// TwinCAT 3 PLC project PlcGenerated
// ProgramVersion: 3.1.4023.0
// libraries:
//   Tc2_Standard, * (Beckhoff Automation GmbH)
//   Tc2_System, * (Beckhoff Automation GmbH)
//   Tc3_Module, * (Beckhoff Automation GmbH)
//   Tc2_EtherCAT,newest,Beckhoff Automation GmbH
// project tree:
//   DUTs/ EthercatDevice.TcDUT
//   / PlcTask.TcTTO
//   POUs/ MAIN.TcPOU
// real-time tasks:
//   TASK PlcTask: cycle T#10ms, priority 20, ADS port 350
// I/O:
//   DEVICE Device_1, AmsNetId 192.168.18.153.2.1
//     Box 1 (LAN9255_EtherCAT_Slave) [LAN9255_EtherCAT_Slave]
// variable links:
//   PlcGenerated/PlcGenerated Instance <-> Device_1/Box 1 (LAN9255_EtherCAT_Slave)
//     PlcTask Inputs/MAIN.DeviceStatus <-> Inputs process data mapping/DeviceStatus
//     PlcTask Inputs/MAIN.MotorDiagnostic <-> Inputs process data mapping/MotorDiagnostic
//     PlcTask Inputs/MAIN.mDiag3 <-> Inputs process data mapping/Diag3
//     PlcTask Inputs/MAIN.mPosition <-> Inputs process data mapping/Position
//     PlcTask Inputs/MAIN.mTemperature <-> Inputs process data mapping/Temperature
//     PlcTask Outputs/MAIN.device[1].mDirection <-> Outputs process data mapping/Direction
//     PlcTask Outputs/MAIN.device[1].mDisplacement <-> Outputs process data mapping/Displacement
//     PlcTask Outputs/MAIN.device[1].mMode <-> Outputs process data mapping/Mode
//     PlcTask Outputs/MAIN.device[1].mRPM <-> Outputs process data mapping/RPM
//     PlcTask Outputs/MAIN.device[1].mRampDelay <-> Outputs process data mapping/RampDelay
//     PlcTask Outputs/MAIN.device[1].mTime <-> Outputs process data mapping/Time

CONFIGURATION PlcGenerated
    RESOURCE PLC ON TwinCAT3
        TASK PlcTask(INTERVAL := T#10ms, PRIORITY := 20);
        PROGRAM MAIN WITH PlcTask : MAIN;
    END_RESOURCE
END_CONFIGURATION

// ---- DUTs/EthercatDevice.TcDUT
TYPE EthercatDevice :
STRUCT
    mDirection AT %Q*: BOOL;
    mRPM AT %Q*: REAL;
    mDisplacement AT %Q*: REAL;
    mTime AT %Q*: REAL;
    mRampDelay AT %Q*: REAL;
    mMode AT %Q*: DWORD;
END_STRUCT
END_TYPE

// ---- POUs/MAIN.TcPOU
PROGRAM MAIN 
VAR CONSTANT 
deviceCount : WORD := 1; 
END_VAR 
VAR 
{attribute 'TcLinkTo' := '[1].mDirection :=  TIID^Device_1^Box 1 (LAN9255_EtherCAT_Slave)^Outputs process data mapping^Direction; 
[1].mDisplacement := TIID^Device_1^Box 1 (LAN9255_EtherCAT_Slave)^Outputs process data mapping^Displacement; 
[1].mRPM := TIID^Device_1^Box 1 (LAN9255_EtherCAT_Slave)^Outputs process data mapping^RPM; 
[1].mTime := TIID^Device_1^Box 1 (LAN9255_EtherCAT_Slave)^Outputs process data mapping^Time; 
[1].mRampDelay := TIID^Device_1^Box 1 (LAN9255_EtherCAT_Slave)^Outputs process data mapping^RampDelay; 
[1].mMode := TIID^Device_1^Box 1 (LAN9255_EtherCAT_Slave)^Outputs process data mapping^Mode'}
device : ARRAY [1..deviceCount] OF EthercatDevice ; 
{attribute 'TcLinkTo' := '[1]:= TIID^Device_1^Box 1 (LAN9255_EtherCAT_Slave)^Inputs process data mapping^Position'}
mPosition AT %I* : ARRAY [1..deviceCount] OF REAL ;
{attribute 'TcLinkTo' := '[1]:= TIID^Device_1^Box 1 (LAN9255_EtherCAT_Slave)^Inputs process data mapping^Temperature'}
mTemperature AT %I* : ARRAY [1..deviceCount] OF DWORD ;
{attribute 'TcLinkTo' := '[1]:=  TIID^Device_1^Box 1 (LAN9255_EtherCAT_Slave)^Inputs process data mapping^MotorDiagnostic'}
MotorDiagnostic AT %I*: ARRAY [1..deviceCount] OF DWORD ;
{attribute 'TcLinkTo' := '[1]:=  TIID^Device_1^Box 1 (LAN9255_EtherCAT_Slave)^Inputs process data mapping^DeviceStatus'}
DeviceStatus AT %I*: ARRAY [1..deviceCount] OF DWORD ;
{attribute 'TcLinkTo' := '[1]:=  TIID^Device_1^Box 1 (LAN9255_EtherCAT_Slave)^Inputs process data mapping^Diag3'}
mDiag3 AT %I*: ARRAY [1..deviceCount] OF DWORD ;
foe_sAmsNetId: T_AmsNetId :='192.168.18.153.2.1';
foe_sAmsPort: ARRAY[1..deviceCount] OF UINT :=[1001];
fbDownload : FB_EcFoeLoad ;
foe_dwPass     : DWORD := 0; // 287454020
foe_nSlaveAddr : UINT := 0;
foe_eMode      : E_EcFoeMode := eFoeMode_Write;
foe_sPathName : STRING := '';
foe_bLoad      : BOOL;
foe_bBusy      : BOOL;
foe_bError     : BOOL;
foe_nErrID     : UDINT;
foe_nBytesWritten : UDINT;
foe_nPercent      : UDINT;

fbSetSlaveState: FB_EcSetSlaveState;
ecs_bExecute   : BOOL; 
ecs_reqState   : WORD; 
ecs_bBusy     : BOOL;
ecs_bError    : BOOL;
ecs_nErrId    : UDINT;
ecs_currState : ST_EcSlaveState;
fbGetSlaveState : FB_EcGetSlaveState;
state           : ST_EcSlaveState;ecg_bExecute : BOOL;ecg_bError          : BOOL;ecg_nErrId          : UDINT;
fbGetAllSlaveStates : FB_EcGetAllSlaveStates;
    ECAbExecute            : BOOL;
    ECAdevStates           : ARRAY[1..deviceCount] OF ST_EcSlaveState;
    ECAnSlaves             : UINT := 0;
    ECAbError              : BOOL;
    ECAnErrId              : UDINT;
END_VAR

fbDownload( bExecute := foe_bLoad,
		sNetId  := foe_sAmsNetId,
		nSlaveAddr := foe_nSlaveAddr,
		dwPass  := foe_dwPass,
		sPathName  := foe_sPathName, 
        bBusy => foe_bBusy,
        bError => foe_bError,
        nErrId => foe_nErrID,
        cbLoad => foe_nBytesWritten,
        nProgress => foe_nPercent );
fbSetSlaveState(
	sNetId := foe_sAmsNetId,
	nSlaveAddr := foe_nSlaveAddr,
	bExecute := ecs_bExecute,
	reqState := ecs_reqState, 
	nErrId =>ecs_nErrId, 
	bBusy=> ecs_bBusy, 
	bError=>ecs_bError
);
fbGetSlaveState(sNetId:= foe_sAmsNetId, nSlaveAddr:= foe_nSlaveAddr, bExecute:=ecg_bExecute);
state := fbGetSlaveState.state;
 ecg_bError := fbGetSlaveState.bError;
 ecg_nErrId := fbGetSlaveState.nErrId;
fbGetAllSlaveStates(sNetId:= foe_sAmsNetId, pStateBuf := ADR(ECAdevStates), cbBufLen:=SIZEOF(ECAdevStates), bExecute:=ECAbExecute);
ECAnSlaves := fbGetAllSlaveStates.nSlaves;
ECAbError := fbGetAllSlaveStates.bError;
ECAnErrId := fbGetAllSlaveStates.nErrId;

END_PROGRAM
